{attribute addProperty BoxType "EK1100-0000-0018"}
{attribute addProperty Id "Beckhoff_EL29xxEK1122Beckhoff_EL29xxEK1122_E909BF84162A_0001_EL2911_0000_0016EL2911_EDE01F6524831A_0002_EL2912_0000_0016EL2912_51553E3C25632"}
{attribute addProperty CRC "1239024676"}
{attribute addProperty SizeInBites "520"}
{attribute addProperty SizeInBytes "65"}
TYPE Beckhoff_EL29xx_49DA0424 EXTENDS EK1100_179A0949 :
STRUCT
	{attribute addProperty Name "Beckhoff_EL29xxEK1122"}
	Beckhoff_EL29xxEK1122 : Beckhoff_EL29xxEK1122_E909BF84;
	{attribute addProperty Name "A_0001_EL2911_0000_0016"}
	A_0001_EL2911_0000_0016 : EL2911_EDE01F65;
	{attribute addProperty Name "A_0002_EL2912_0000_0016"}
	A_0002_EL2912_0000_0016 : EL2912_51553E3C;
END_STRUCT
END_TYPE

(* stored: Version 1.2.0.0, ProductVersion 3.1.4024.9
   DUT Beckhoff_EL29xx_49DA0424: Id {9b8d986c-c571-41a8-b3dd-660189b87f4c} *)
